# EPICS substitutions: ek9000App/Db/EL4014.substitutions
file EL4014.template
{       pattern
        {
                TERMINAL,

        }
        {
        }
}
